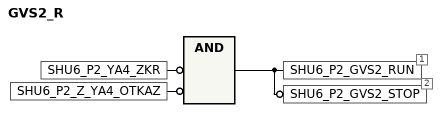
_CFC_ (* Continuous Function Chart, elements in execution order *)
#0 AND(NOT SHU6_P2_YA4_ZKR, NOT SHU6_P2_Z_YA4_OTKAZ)
#1 SHU6_P2_GVS2_RUN <= #0
#2 SHU6_P2_GVS2_STOP <= NOT #0
_END_CFC_
END_PROGRAM

(* POU TZBiS/S/HVS_R, CFC *)
PROGRAM HVS_R
VAR
END_VAR
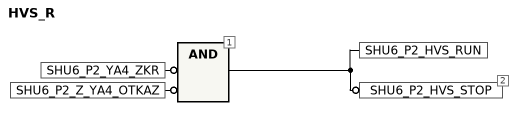
_CFC_ (* Continuous Function Chart, elements in execution order *)
#0 SHU6_P2_HVS_RUN <= #1
#1 AND(NOT SHU6_P2_YA4_ZKR, NOT SHU6_P2_Z_YA4_OTKAZ)
#2 SHU6_P2_HVS_STOP <= NOT #1
_END_CFC_
END_PROGRAM

(* POU TZBiS/S/S_STER_REG, CFC *)
PROGRAM S_STER_REG
VAR
	ZAD_S_Ster_Reg: TON;
END_VAR
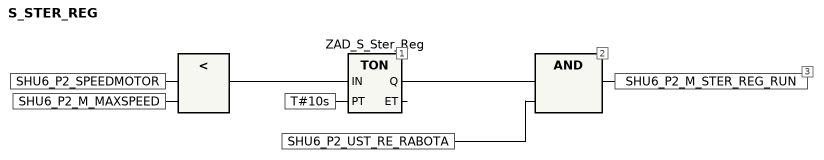
_CFC_ (* Continuous Function Chart, elements in execution order *)
#0 <(SHU6_P2_SPEEDMOTOR, SHU6_P2_M_MAXSPEED)
#1 ZAD_S_Ster_Reg:TON(IN: #0, PT: T#10s)
#2 AND(#1.Q, SHU6_P2_UST_RE_RABOTA)
#3 SHU6_P2_M_STER_REG_RUN <= #2
_END_CFC_
END_PROGRAM

(* POU TZBiS/S/S_ZAM, CFC *)
PROGRAM S_ZAM
VAR
	SR_ZAM: SR;
END_VAR
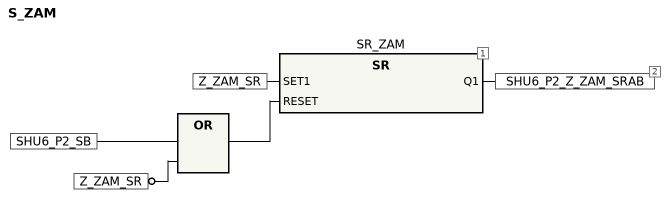
_CFC_ (* Continuous Function Chart, elements in execution order *)
#0 OR(SHU6_P2_SB, NOT Z_ZAM_SR)
#1 SR_ZAM:SR(SET1: Z_ZAM_SR, RESET: #0)
#2 SHU6_P2_Z_ZAM_SRAB <= #1.Q1
_END_CFC_
(* the same logic as Structured Text *)
SR_ZAM(SET1 := Z_ZAM_SR, RESET := SHU6_P2_SB OR NOT Z_ZAM_SR);
SHU6_P2_Z_ZAM_SRAB := SR_ZAM.Q1;
END_PROGRAM

(* POU TZBiS/TZB/Z_FC_NPit, CFC *)
PROGRAM Z_FC_NPit
VAR
	SR_YA1_YA2_NPit: SR;
	SR_IBP_NPit: SR;
	SR_A1_G1_NPit: SR;
	SR_A1_TV1_NPit: SR;
	SR_24V_NPit: SR;
END_VAR
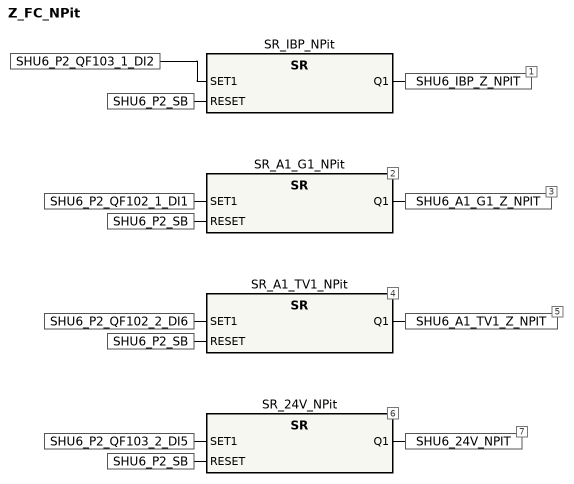
_CFC_ (* Continuous Function Chart, elements in execution order *)
#0 SR_IBP_NPit:SR(SET1: SHU6_P2_QF103_1_DI2, RESET: SHU6_P2_SB)
#1 SHU6_IBP_Z_NPIT <= #0.Q1
#2 SR_A1_G1_NPit:SR(SET1: SHU6_P2_QF102_1_DI1, RESET: SHU6_P2_SB)
#3 SHU6_A1_G1_Z_NPIT <= #2.Q1
#4 SR_A1_TV1_NPit:SR(SET1: SHU6_P2_QF102_2_DI6, RESET: SHU6_P2_SB)
#5 SHU6_A1_TV1_Z_NPIT <= #4.Q1
#6 SR_24V_NPit:SR(SET1: SHU6_P2_QF103_2_DI5, RESET: SHU6_P2_SB)
#7 SHU6_24V_NPIT <= #6.Q1
_END_CFC_
(* the same logic as Structured Text *)
SR_IBP_NPit(SET1 := SHU6_P2_QF103_1_DI2, RESET := SHU6_P2_SB);
SHU6_IBP_Z_NPIT := SR_IBP_NPit.Q1;
SR_A1_G1_NPit(SET1 := SHU6_P2_QF102_1_DI1, RESET := SHU6_P2_SB);
SHU6_A1_G1_Z_NPIT := SR_A1_G1_NPit.Q1;
SR_A1_TV1_NPit(SET1 := SHU6_P2_QF102_2_DI6, RESET := SHU6_P2_SB);
SHU6_A1_TV1_Z_NPIT := SR_A1_TV1_NPit.Q1;
SR_24V_NPit(SET1 := SHU6_P2_QF103_2_DI5, RESET := SHU6_P2_SB);
SHU6_24V_NPIT := SR_24V_NPit.Q1;
END_PROGRAM

(* POU TZBiS/TZB/ALL_TZB, CFC *)
PROGRAM ALL_TZB
VAR
END_VAR
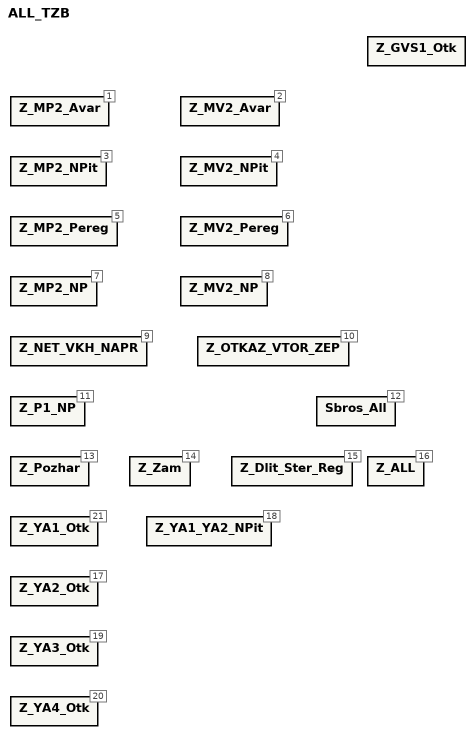
_CFC_ (* Continuous Function Chart, elements in execution order *)
#0 Z_GVS1_Otk()
#1 Z_MP2_Avar()
#2 Z_MV2_Avar()
#3 Z_MP2_NPit()
#4 Z_MV2_NPit()
#5 Z_MP2_Pereg()
#6 Z_MV2_Pereg()
#7 Z_MP2_NP()
#8 Z_MV2_NP()
#9 Z_NET_VKH_NAPR()
#10 Z_OTKAZ_VTOR_ZEP()
#11 Z_P1_NP()
#12 Sbros_All()
#13 Z_Pozhar()
#14 Z_Zam()
#15 Z_Dlit_Ster_Reg()
#16 Z_ALL()
#17 Z_YA2_Otk()
#18 Z_YA1_YA2_NPit()
#19 Z_YA3_Otk()
#20 Z_YA4_Otk()
#21 Z_YA1_Otk()
_END_CFC_
(* the same logic as Structured Text *)
Z_GVS1_Otk();
Z_MP2_Avar();
Z_MV2_Avar();
Z_MP2_NPit();
Z_MV2_NPit();
Z_MP2_Pereg();
Z_MV2_Pereg();
Z_MP2_NP();
Z_MV2_NP();
Z_NET_VKH_NAPR();
Z_OTKAZ_VTOR_ZEP();
Z_P1_NP();
Sbros_All();
Z_Pozhar();
Z_Zam();
Z_Dlit_Ster_Reg();
Z_ALL();
Z_YA2_Otk();
Z_YA1_YA2_NPit();
Z_YA3_Otk();
Z_YA4_Otk();
Z_YA1_Otk();
END_PROGRAM

(* POU TZBiS/TZB/Z_GVS1_Otk, CFC *)
PROGRAM Z_GVS1_Otk
VAR
	TON_YA3_OTKAZ: TON;
	SR_GVS1_Otkaz: SR;
	TON_YA3_Z_ZAM: TON;
END_VAR
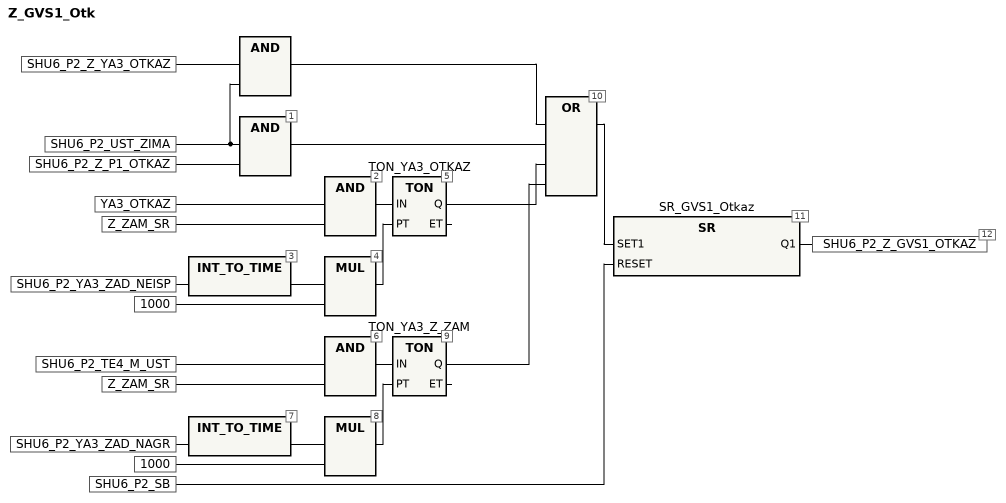
_CFC_ (* Continuous Function Chart, elements in execution order *)
#0 AND(SHU6_P2_Z_YA3_OTKAZ, SHU6_P2_UST_ZIMA)
#1 AND(SHU6_P2_UST_ZIMA, SHU6_P2_Z_P1_OTKAZ)
#2 AND(YA3_OTKAZ, Z_ZAM_SR)
#3 INT_TO_TIME(SHU6_P2_YA3_ZAD_NEISP)
#4 MUL(#3, 1000)
#5 TON_YA3_OTKAZ:TON(IN: #2, PT: #4)
#6 AND(SHU6_P2_TE4_M_UST, Z_ZAM_SR)
#7 INT_TO_TIME(SHU6_P2_YA3_ZAD_NAGR)
#8 MUL(#7, 1000)
#9 TON_YA3_Z_ZAM:TON(IN: #6, PT: #8)
#10 OR(#0, #1, #5.Q, #9.Q)
#11 SR_GVS1_Otkaz:SR(SET1: #10, RESET: SHU6_P2_SB)
#12 SHU6_P2_Z_GVS1_OTKAZ <= #11.Q1
_END_CFC_
(* the same logic as Structured Text *)
TON_YA3_OTKAZ(IN := YA3_OTKAZ AND Z_ZAM_SR, PT := INT_TO_TIME(SHU6_P2_YA3_ZAD_NEISP) * 1000);
TON_YA3_Z_ZAM(IN := SHU6_P2_TE4_M_UST AND Z_ZAM_SR, PT := INT_TO_TIME(SHU6_P2_YA3_ZAD_NAGR) * 1000);
SR_GVS1_Otkaz(SET1 := (SHU6_P2_Z_YA3_OTKAZ AND SHU6_P2_UST_ZIMA) OR (SHU6_P2_UST_ZIMA AND SHU6_P2_Z_P1_OTKAZ) OR TON_YA3_OTKAZ.Q OR TON_YA3_Z_ZAM.Q, RESET := SHU6_P2_SB);
SHU6_P2_Z_GVS1_OTKAZ := SR_GVS1_Otkaz.Q1;
END_PROGRAM

(* POU TZBiS/TZB/Z_MP2/Z_MP2_Avar, CFC *)
PROGRAM Z_MP2_Avar
VAR
	SR_MP2_Avar: SR;
	SR_MP2R_Avar: SR;
	TON_ALM_DI3: TON;
END_VAR
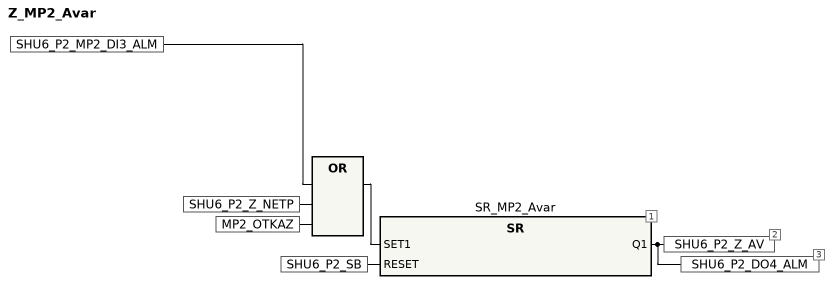
_CFC_ (* Continuous Function Chart, elements in execution order *)
#0 OR(SHU6_P2_MP2_DI3_ALM, SHU6_P2_Z_NETP, MP2_OTKAZ)
#1 SR_MP2_Avar:SR(SET1: #0, RESET: SHU6_P2_SB)
#2 SHU6_P2_Z_AV <= #1.Q1
#3 SHU6_P2_DO4_ALM <= #1.Q1
_END_CFC_
(* the same logic as Structured Text *)
SR_MP2_Avar(SET1 := SHU6_P2_MP2_DI3_ALM OR SHU6_P2_Z_NETP OR MP2_OTKAZ, RESET := SHU6_P2_SB);
SHU6_P2_Z_AV := SR_MP2_Avar.Q1;
SHU6_P2_DO4_ALM := SR_MP2_Avar.Q1;
END_PROGRAM

(* POU TZBiS/TZB/Z_MV2/Z_MV2_Avar, CFC *)
PROGRAM Z_MV2_Avar
VAR
	SR_MV2_Avar: SR;
	SR_MV2R_Avar: SR;
	TON_ALM_DI4: TON;
END_VAR
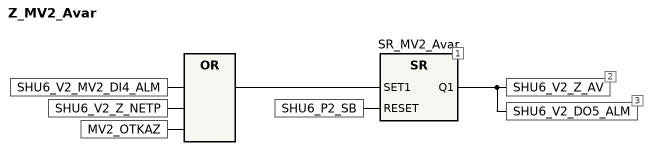
_CFC_ (* Continuous Function Chart, elements in execution order *)
#0 OR(SHU6_V2_MV2_DI4_ALM, SHU6_V2_Z_NETP, MV2_OTKAZ)
#1 SR_MV2_Avar:SR(SET1: #0, RESET: SHU6_P2_SB)
#2 SHU6_V2_Z_AV <= #1.Q1
#3 SHU6_V2_DO5_ALM <= #1.Q1
_END_CFC_
(* the same logic as Structured Text *)
SR_MV2_Avar(SET1 := SHU6_V2_MV2_DI4_ALM OR SHU6_V2_Z_NETP OR MV2_OTKAZ, RESET := SHU6_P2_SB);
SHU6_V2_Z_AV := SR_MV2_Avar.Q1;
SHU6_V2_DO5_ALM := SR_MV2_Avar.Q1;
END_PROGRAM

(* POU TZBiS/TZB/Z_MP2/Z_MP2_NPit, CFC *)
PROGRAM Z_MP2_NPit
VAR
	SR_MP2_NPit: SR;
	SR_M4_6R_NPit: SR;
END_VAR
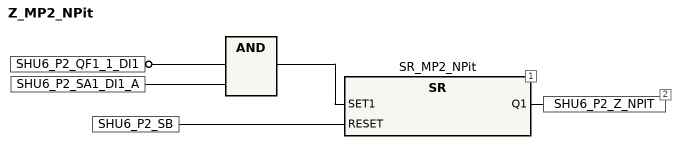
_CFC_ (* Continuous Function Chart, elements in execution order *)
#0 AND(NOT SHU6_P2_QF1_1_DI1, SHU6_P2_SA1_DI1_A)
#1 SR_MP2_NPit:SR(SET1: #0, RESET: SHU6_P2_SB)
#2 SHU6_P2_Z_NPIT <= #1.Q1
_END_CFC_
(* the same logic as Structured Text *)
SR_MP2_NPit(SET1 := NOT SHU6_P2_QF1_1_DI1 AND SHU6_P2_SA1_DI1_A, RESET := SHU6_P2_SB);
SHU6_P2_Z_NPIT := SR_MP2_NPit.Q1;
END_PROGRAM

(* POU TZBiS/TZB/Z_MV2/Z_MV2_NPit, CFC *)
PROGRAM Z_MV2_NPit
VAR
	SR_MV2_NPit: SR;
	SR_MV2R_NPit: SR;
END_VAR
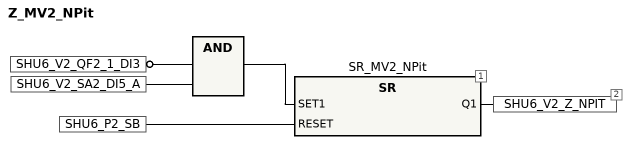
_CFC_ (* Continuous Function Chart, elements in execution order *)
#0 AND(NOT SHU6_V2_QF2_1_DI3, SHU6_V2_SA2_DI5_A)
#1 SR_MV2_NPit:SR(SET1: #0, RESET: SHU6_P2_SB)
#2 SHU6_V2_Z_NPIT <= #1.Q1
_END_CFC_
(* the same logic as Structured Text *)
SR_MV2_NPit(SET1 := NOT SHU6_V2_QF2_1_DI3 AND SHU6_V2_SA2_DI5_A, RESET := SHU6_P2_SB);
SHU6_V2_Z_NPIT := SR_MV2_NPit.Q1;
END_PROGRAM

(* POU TZBiS/TZB/Z_MP2/Z_MP2_Pereg, CFC *)
PROGRAM Z_MP2_Pereg
VAR
	SR_SHU6_P2_TSMP2_DI1: SR;
	TOF_TSMP1: TOF;
	TON1: TON;
	SR_SHU6_P2R_TSMP2R_DI2:SR;
	TOF_TSMP2 :TOF;
	TON2: TON;
END_VAR
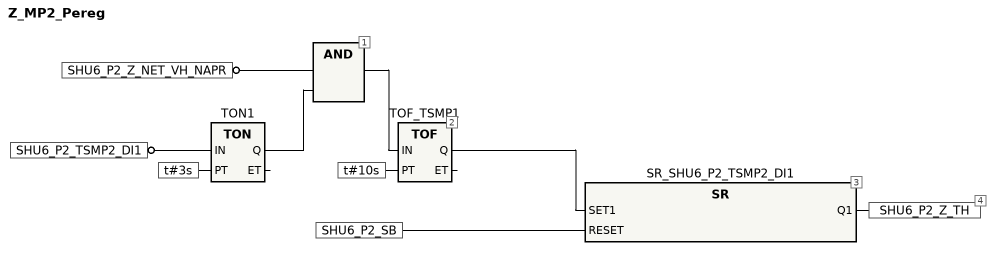
_CFC_ (* Continuous Function Chart, elements in execution order *)
#0 TON1:TON(IN: NOT SHU6_P2_TSMP2_DI1, PT: t#3s)
#1 AND(NOT SHU6_P2_Z_NET_VH_NAPR, #0.Q)
#2 TOF_TSMP1:TOF(IN: #1, PT: t#10s)
#3 SR_SHU6_P2_TSMP2_DI1:SR(SET1: #2.Q, RESET: SHU6_P2_SB)
#4 SHU6_P2_Z_TH <= #3.Q1
_END_CFC_
(* the same logic as Structured Text *)
TON1(IN := NOT SHU6_P2_TSMP2_DI1, PT := t#3s);
TOF_TSMP1(IN := NOT SHU6_P2_Z_NET_VH_NAPR AND TON1.Q, PT := t#10s);
SR_SHU6_P2_TSMP2_DI1(SET1 := TOF_TSMP1.Q, RESET := SHU6_P2_SB);
SHU6_P2_Z_TH := SR_SHU6_P2_TSMP2_DI1.Q1;
END_PROGRAM

(* POU TZBiS/TZB/Z_MV2/Z_MV2_Pereg, CFC *)
PROGRAM Z_MV2_Pereg
VAR
	TON2:TON;
	TOF_TSMP2: TOF;
	TON1: TON;
	TOF_TSMV1: TOF;
	TOF_TSMV2: TOF;
	SR_SHU6_P2_TSMV2_DI1: SR;
	SR_SHU6_P2R_TSMV2R_DI2: SR;
END_VAR
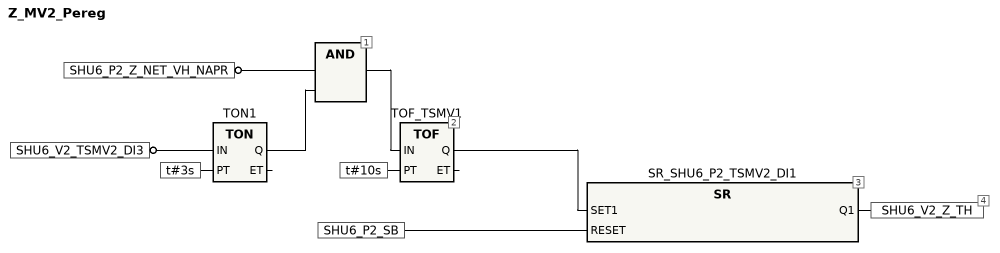
_CFC_ (* Continuous Function Chart, elements in execution order *)
#0 TON1:TON(IN: NOT SHU6_V2_TSMV2_DI3, PT: t#3s)
#1 AND(NOT SHU6_P2_Z_NET_VH_NAPR, #0.Q)
#2 TOF_TSMV1:TOF(IN: #1, PT: t#10s)
#3 SR_SHU6_P2_TSMV2_DI1:SR(SET1: #2.Q, RESET: SHU6_P2_SB)
#4 SHU6_V2_Z_TH <= #3.Q1
_END_CFC_
(* the same logic as Structured Text *)
TON1(IN := NOT SHU6_V2_TSMV2_DI3, PT := t#3s);
TOF_TSMV1(IN := NOT SHU6_P2_Z_NET_VH_NAPR AND TON1.Q, PT := t#10s);
SR_SHU6_P2_TSMV2_DI1(SET1 := TOF_TSMV1.Q, RESET := SHU6_P2_SB);
SHU6_V2_Z_TH := SR_SHU6_P2_TSMV2_DI1.Q1;
END_PROGRAM

(* POU TZBiS/TZB/Z_MP2/Z_MP2_NP, CFC *)
PROGRAM Z_MP2_NP
VAR
	TON_PDS2: TON;
	TON_ReRab: TON;
	TON_MVKL: TON;
	TON_AVT: TON;
	TP_SR: TP;
	SR_NP_M1: SR;
	SR_NP_M2: SR;
	TON_MVKL_M1: TON;
	TON_AVT_M1: TON;
	TON_AVT_M2: TON;
	TON_MVKL_M2: TON;
END_VAR
